PROGRAM MAIN
VAR
	fbSuperBohrmachine: SuperBohrmachine;
END_VAR

fbSuperBohrmachine();

END_PROGRAM

(* stored: Version 1.1.0.1, ProductVersion 3.1.4024.3
   POU MAIN: Id {fd9c62c6-08ad-42ca-a926-6612bb53b12d}, SpecialFunc None *)
